(* IEC 61131-3 sources: Lasal/CPU_5344_V01/Class/Logic_And_2, 1 file *)

(* ---- Logic_And_2.st ---- *)
(*!
<Class
	Name               = "Logic_And_2"
	Revision           = "1.2"
	RealtimeTask       = "false"
	CyclicTask         = "false"
	BackgroundTask     = "false"
	Sigmatek           = "true"
	OSInterface        = "false"
	HighPriority       = "false"
	Automatic          = "false"
	UpdateMode         = "Prescan"
	IconPath           = ".\Class\Logic_And_2\Logic_And_Base.ico"
	SharedCommandTable = "true"
	Objectsize         = "(284,120)"
	Comment            = "V1.2 Logic AND class with 2 operands">
	<Channels>
		<Server
			Name           = "result"
			Initialize     = "false"
			Visualized     = "true"
			WriteProtected = "true"
			Comment        = "if all operands are &lt;&gt; 0 then result = 1 ">
		</Server>
		<Client Name="Op1" Required="false" Internal="false" Comment="Operand 1"/>
		<Client Name="Op2" Required="false" Internal="false" Comment="Operand 2"/>
	</Channels>
	<Network Name="Logic_And_2">
		<!-- List of Components in this network -->
		<Components>
			<Object
				Name       = "_base"
				Class      = "Logic_And_Base"
				Position   = "(630,450)"
				Visualized = "true">
				<Channels>
					<Server Name="result"/>
				</Channels>
			</Object>
		</Components>
		<Comments>
		</Comments>
		<!-- List of Connections in this network -->
		<Connections>
			<Connection Source="this.result" Destination="_base.result" Vertices="(1102,210),(930,540),"/>
		</Connections>
		<!-- Headerfiles -->
		<Options>
		</Options>
	</Network>
</Class>
*)
#pragma using Logic_And_Base

Logic_And_2 : CLASS
: Logic_And_Base
  //Servers:
  //Clients:
	Op1 	: CltCh_DINT;
	Op2 	: CltCh_DINT;
  //Variables:
  //Functions:
  //Tables:
	FUNCTION @STD
		VAR_OUTPUT
			ret_code	: CONFSTATES;
		END_VAR;
	FUNCTION GLOBAL TAB @CT_;
END_CLASS;
